TYPE ST_Sts_PlcComOut :
STRUCT
	bUnderLight			: BOOL;
	bGripper			: BOOL;
	bPusher				: BOOL;
	bHeaterFan			: BOOL;
	bHeaterElement		: BOOL;
END_STRUCT
END_TYPE

(* stored: Version 1.1.0.1
   DUT ST_Sts_PlcComOut: Id {c451a995-5e6c-4b37-9b64-162fb8e09a61} *)
